// Mitsubishi GX Works2 project: fx3U-48MT_blink_byone   PLC: FX3U/FX3UC

PROGRAM MAIN
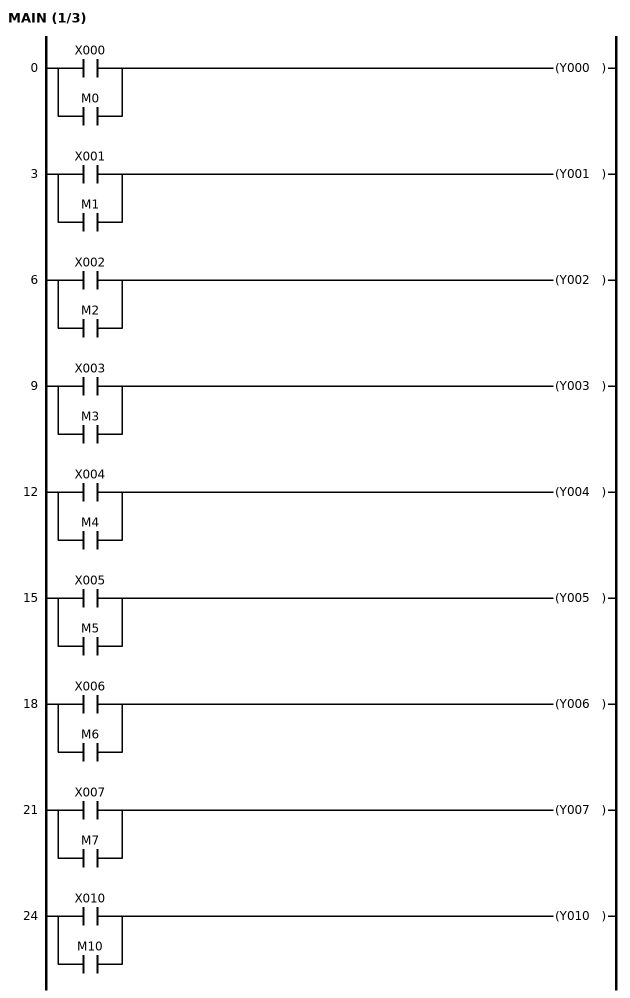
0     LD      X000
      OR      M0
      OUT     Y000
3     LD      X001
      OR      M1
      OUT     Y001
6     LD      X002
      OR      M2
      OUT     Y002
9     LD      X003
      OR      M3
      OUT     Y003
12    LD      X004
      OR      M4
      OUT     Y004
15    LD      X005
      OR      M5
      OUT     Y005
18    LD      X006
      OR      M6
      OUT     Y006
21    LD      X007
      OR      M7
      OUT     Y007
24    LD      X010
      OR      M10
      OUT     Y010
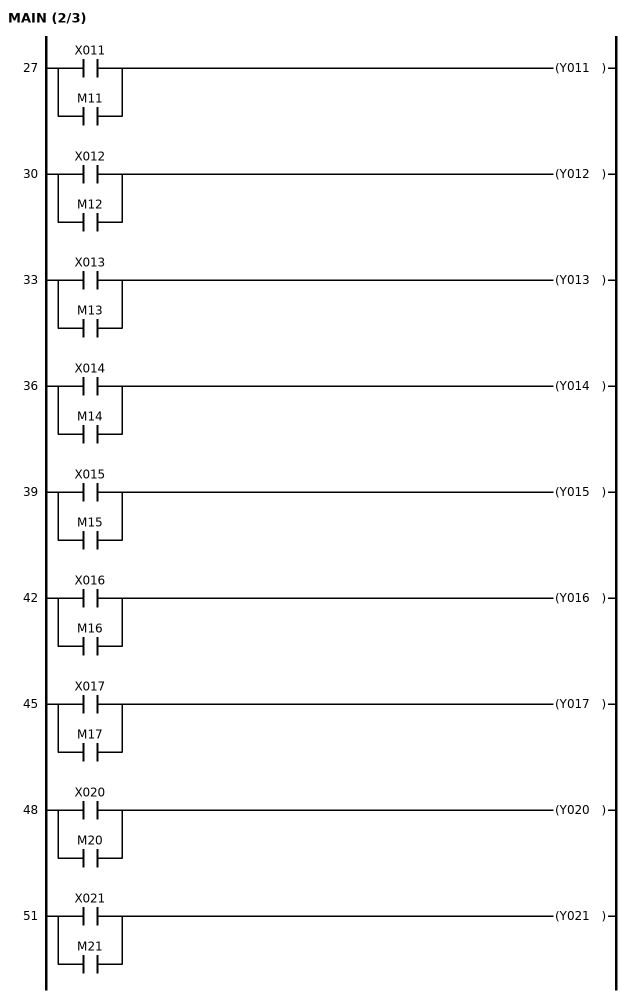
27    LD      X011
      OR      M11
      OUT     Y011
30    LD      X012
      OR      M12
      OUT     Y012
33    LD      X013
      OR      M13
      OUT     Y013
36    LD      X014
      OR      M14
      OUT     Y014
39    LD      X015
      OR      M15
      OUT     Y015
42    LD      X016
      OR      M16
      OUT     Y016
45    LD      X017
      OR      M17
      OUT     Y017
48    LD      X020
      OR      M20
      OUT     Y020
51    LD      X021
      OR      M21
      OUT     Y021
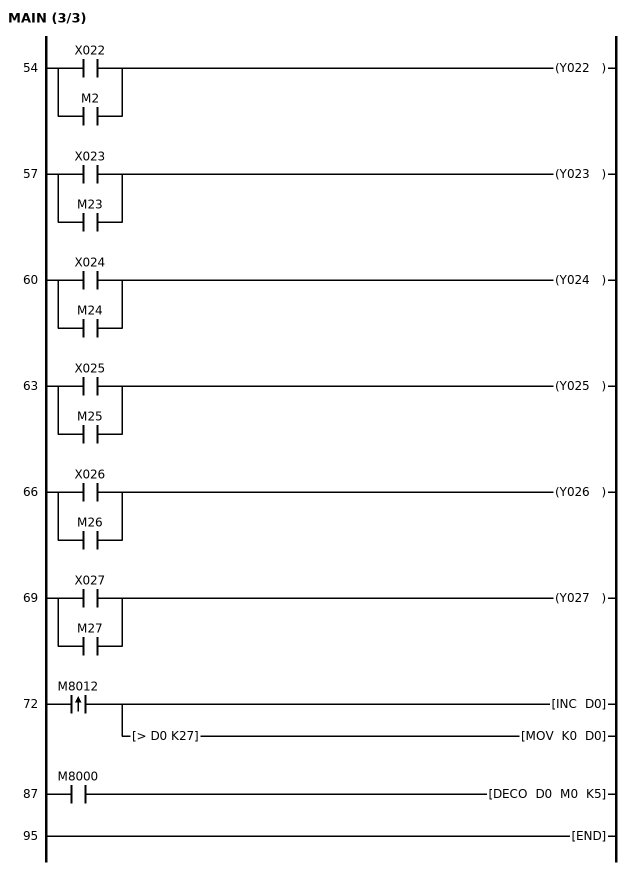
54    LD      X022
      OR      M2
      OUT     Y022
57    LD      X023
      OR      M23
      OUT     Y023
60    LD      X024
      OR      M24
      OUT     Y024
63    LD      X025
      OR      M25
      OUT     Y025
66    LD      X026
      OR      M26
      OUT     Y026
69    LD      X027
      OR      M27
      OUT     Y027
72    LDP     M8012
      INC     D0
      AND>    D0 K27
      MOV     K0 D0
87    LD      M8000
      DECO    D0 M0 K5
95    END
END_PROGRAM
